{attribute 'GeneratedUsingTerminal: KL2642-0050'}
{attribute addProperty BoxType "KL2642-0050"}
{attribute addProperty Id "State_RelayAT %I*BOOL0OutputAT %Q*BOOL0"}
{attribute addProperty CRC "4124805841"}
{attribute addProperty Size "0"}
TYPE Channel_F5DB8AD1 :
STRUCT
	{attribute addProperty Name "State_Relay"}
	State_Relay AT %I* : BOOL;
	{attribute addProperty Name "Output"}
	Output AT %Q* : BOOL;
END_STRUCT
END_TYPE
